gfCNCPoint4[29977] = {X 172.8551, Y 45.0534, Z -6.3333, A 0.000, B 0.000, C 0.000 }
gfCNCPoint4[29978] = {X 171.8455, Y 43.8849, Z -6.3333, A 0.000, B 0.000, C 0.000 }
gfCNCPoint4[29979] = {X 170.9813, Y 42.6051, Z -6.3333, A 0.000, B 0.000, C 0.000 }
gfCNCPoint4[29980] = {X 170.2746, Y 41.2320, Z -6.3333, A 0.000, B 0.000, C 0.000 }
gfCNCPoint4[29981] = {X 169.7354, Y 39.7849, Z -6.3333, A 0.000, B 0.000, C 0.000 }
gfCNCPoint4[29982] = {X 169.3712, Y 38.2842, Z -6.3333, A 0.000, B 0.000, C 0.000 }
gfCNCPoint4[29983] = {X 169.3156, Y 37.9356, Z -6.3333, A 0.000, B 0.000, C 0.000 }
gfCNCPoint4[29984] = {X 165.3654, Y 38.5645, Z -6.3333, A 0.000, B 0.000, C 0.000 }
gfCNCPoint4[29985] = {X 169.3946, Y 37.9230, Z -6.3333, A 0.000, B 0.000, C 0.000 }
gfCNCPoint4[29986] = {X 169.3392, Y 37.5748, Z -6.3333, A 0.000, B 0.000, C 0.000 }
gfCNCPoint4[29987] = {X 169.1819, Y 35.9788, Z -6.3333, A 0.000, B 0.000, C 0.000 }
gfCNCPoint4[29988] = {X 169.1989, Y 34.3752, Z -6.3333, A 0.000, B 0.000, C 0.000 }
gfCNCPoint4[29989] = {X 169.3900, Y 32.7829, Z -6.3333, A 0.000, B 0.000, C 0.000 }
gfCNCPoint4[29990] = {X 169.7529, Y 31.2208, Z -6.3333, A 0.000, B 0.000, C 0.000 }
gfCNCPoint4[29991] = {X 170.2834, Y 29.7074, Z -6.3333, A 0.000, B 0.000, C 0.000 }
gfCNCPoint4[29992] = {X 170.9352, Y 28.3792, Z -6.3333, A 0.000, B 0.000, C 0.000 }
gfCNCPoint4[29993] = {X 171.7628, Y 27.1528, Z -6.3333, A 0.000, B 0.000, C 0.000 }
gfCNCPoint4[29994] = {X 172.7505, Y 26.0513, Z -6.3333, A 0.000, B 0.000, C 0.000 }
gfCNCPoint4[29995] = {X 173.8798, Y 25.0955, Z -6.3333, A 0.000, B 0.000, C 0.000 }
gfCNCPoint4[29996] = {X 175.1294, Y 24.3034, Z -6.3333, A 0.000, B 0.000, C 0.000 }
gfCNCPoint4[29997] = {X 174.3081, Y 23.9332, Z -6.3333, A 0.000, B 0.000, C 0.000 }
gfCNCPoint4[29998] = {X 173.5835, Y 23.3979, Z -6.3333, A 0.000, B 0.000, C 0.000 }
gfCNCPoint4[29999] = {X 172.9884, Y 22.7215, Z -6.3333, A 0.000, B 0.000, C 0.000 }
gfCNCPoint4[30000] = {X 172.5496, Y 21.9347, Z -6.3333, A 0.000, B 0.000, C 0.000 }

ENDDAT
